PROGRAM MAIN
VAR
	nCycleCount	: UDINT;
	nIdx		: INT;
	fScaled		: LREAL;
END_VAR

nCycleCount := nCycleCount + 1;

GVL_System.fbCylinder.Cyclic();
GVL_System.fbStation.Cyclic();
GVL_System.fbDerived.Cyclic();

GVL_Hmi.bEnable := (GVL_System.fbStation.State = E_StationState.Running);

fScaled := F_Scale(fValue := 5.0, fMin := 0.0, fMax := 10.0);
GVL_Hmi.nSpeed := LREAL_TO_INT(fScaled * 100.0);

FOR nIdx := 0 TO 9 DO
	GVL_Hmi.arValues[nIdx] := GVL_Hmi.nSpeed;
END_FOR

END_PROGRAM

(* stored: Version 1.1.0.1, ProductVersion 3.1.4024.12
   POU MAIN: Id {29aab4ab-3dcf-4a7e-a966-3622bf8d4b97}, SpecialFunc None *)
